// TIA Portal project "FullDemo" (V17)

(* hardware
DEVICE "S71500/ET200MP station_1"  S7-1500 station
   slot 0: "Rail_0"  Rack  6ES7 590-1***0-0AA0
   slot 0: "PM 70W 120/230VAC"  PM 70W 120/230VAC  6EP1332-4BA00
   slot 1: "S7-1500"  CPU 1513F-1 PN  6ES7 513-1FL01-0AB0  V2.0
      slot 3: "CPU display_1"  6ES7591-1AA00-0AA0
   slot 2: "DI 32x24VDC HF_1"  DI 32x24VDC HF  6ES7 521-1BL00-0AB0  V2.0
   slot 3: "DQ 32x24VDC/0.5A ST_1"  DQ 32x24VDC/0.5A ST  6ES7 522-1BL00-0AB0  V2.0
   slot 4: "AI 8xU/I/RTD/TC ST_1"  AI 8xU/I/RTD/TC ST  6ES7 531-7KF00-0AB0  V2.0
*)

// ===== PLC "S7-1500"  CPU 1513F-1 PN =====
// protected blocks, not shown: "FC_Signal"

VAR_GLOBAL   // PLC tag table "Default tag table"
   "Clock_Byte" AT %MB10 : Byte;
   "Clock_10Hz" AT %M10.0 : Bool;
   "Clock_5Hz" AT %M10.1 : Bool;
   "Clock_2.5Hz" AT %M10.2 : Bool;
   "Clock_2Hz" AT %M10.3 : Bool;
   "Clock_1.25Hz" AT %M10.4 : Bool;
   "Clock_1Hz" AT %M10.5 : Bool;
   "Clock_0.625Hz" AT %M10.6 : Bool;
   "Clock_0.5Hz" AT %M10.7 : Bool;
END_VAR

VAR_GLOBAL   // PLC tag table "Conveyor"
   "B_LB" AT %I4.0 : Bool;   // Lichtschranke / Light barrier
   "S_Bay1" AT %I4.1 : Bool;   // Taster Platz 1 / Momentary contact Bay 1
   "S_Bay2" AT %I4.2 : Bool;   // Taster Platz 2 / Momentary contact Bay 2
   "S_Bay3" AT %I4.3 : Bool;   // Taster Platz 3 / Momentary contact Bay 3
   "S_BayLB" AT %I4.4 : Bool;   // Taster Lichtschranken-Platz / Momentary contact Light barrier bay
   "B_Bay1" AT %I4.5 : Bool;   // Initiator Platz 1 / Proximity sensor Bay 1
   "B_Bay2" AT %I4.6 : Bool;   // Initiator Platz 2 / Proximity sensor Bay 2
   "B_Bay3" AT %I4.7 : Bool;   // Initiator Platz 3 / Proximity sensor Bay 3
   "P_Bay1" AT %Q4.1 : Bool;   // Meldeleuchte Platz 1 / Indicator light Bay 1
   "P_Bay2" AT %Q4.2 : Bool;   // Meldeleuchte Platz 2 / Indicator light Bay 2
   "P_Bay3" AT %Q4.3 : Bool;   // Meldeleuchte Platz 3 / Indicator light Bay 3
   "P_BayLB" AT %Q4.4 : Bool;   // Meldeleuchte Lichtschranken-Platz / Indicator light Light barrier bay
   "K_Right" AT %Q4.5 : Bool;   // Bandmotor Rechts / Run conveyor RIGHT
   "K_Left" AT %Q4.6 : Bool;   // Bandmotor Links / Run conveyor LEFT
   "P_Horn" AT %Q4.7 : Bool;   // Hupe / Horn
END_VAR

VAR_GLOBAL   // PLC tag table "My_Tags"
   "M_AuxLB" AT %M16.0 : Bool;   // Edge auxiliary memory bit Light barrier / Flanken-Hilfsmerker Lichtschranke
   "S_Fault3" AT %E0.6 : Bool;   // Schalter Störung 3 / S_Fault3
   "M_JogRight" AT %M16.2 : Bool;   // Merker Tippen Rechts / Memory bit Jog conveyor RIGHT
   "M_AutoRight" AT %M16.4 : Bool;   // Merker Auto Rechts / Memory bit Conveyor AUTO RIGHT
   "M_ConvFault" AT %M17.0 : Bool;   // Merker Bandlauf-Störung / Memory bit Conveyor fault
   "S_Acknowledge" AT %E0.7 : Bool;   // Taster Quittierung / S_Acknowledge
   "P_Operation" AT %A0.1 : Bool;   // Meldeleuchte Betrieb EIN / Indicator light Operation ON
   "P_Fault" AT %A0.7 : Bool;   // Anzeige Band-Störung / Indicator light for fault
   "M_AuxFault1" AT %M17.1 : Bool;   // Edge auxiliary memory bit Fault 1 / Flanken-Hilfsmerker Störung 1
   "P_Fault1" AT %A0.2 : Bool;   // Anzeige Störung 1 / Indicator light for fault1
   "P_Fault2" AT %A0.3 : Bool;   // Anzeige Störung 2 / Indicator light for fault2
   "S_Fault1" AT %E0.4 : Bool;   // Schalter Störung 1 / S_Fault1
   "S_Fault2" AT %E0.5 : Bool;   // Schalter Störung 2 / S_Fault2
   "P_Fault3" AT %A0.4 : Bool;   // Anzeige Störung 3 / Indicator light for fault3
   "M_AuxOpON" AT %M15.1 : Bool;   // Edge auxiliary memory bit Operation ON / Flanken-Hilfsmerker Anlage EIN
   "M_ActSetp" AT %M18.4 : Bool;   // Merker Ist-Stückzahl=Soll-Stückzah / Memory bit Actual- has reached Setpoint number
   "S_OperationON" AT %E0.1 : Bool;   // Taster Betrieb EIN / S_OperationON
   "S_OperationOFF" AT %E0.0 : Bool;   // Taster Betrieb AUS / S_OperationOFF
   "S_Right" AT %E0.2 : Bool;   // Taster Tippen Rechts / S_Right
   "S_Left" AT %E0.3 : Bool;   // Taster Tippen Links / S_Left
   "M_StorFault1" AT %M17.2 : Bool;   // Memory bit for storing Fault 1 / Merker Meldespeicher Störung 1
   "M_AuxFault2" AT %M17.3 : Bool;   // Edge auxiliary memory bit Fault 2 / Flanken-Hilfsmerker Störung 2
   "M_StorFault2" AT %M17.4 : Bool;   // Memory bit for storing Fault 2 / Merker Meldespeicher Störung 2
   "TOF-Timer-L" AT %M20.2 : Bool;
   "TOF-Timer-R" AT %M20.1 : Bool;
   "max_ConvFault" AT %M20.0 : Bool;
   "P_InitLeft" AT %A0.5 : Bool;
   "P_InitRight" AT %A0.6 : Bool;
   "S_Slider1" AT %IW10 : Word;
   "S_Slider2" AT %IW30 : Word;
END_VAR

VAR_GLOBAL CONSTANT   // PLC tag table "My_Tags"
   "const_maxTime" : Time := t#6s;   // max. Transportzeit / max. transport time
   "const_Setp" : UInt := 3;   // Sollwert / setpoint parts
END_VAR

VAR_GLOBAL   // PLC tag table "Drive"
   "StatusWordDrive" AT %EW60 : Word;
   "ActualSpeedDrive" AT %EW62 : Int;
   "ControlWordDrive" AT %AW60 : Word;
   "SetPointSpeedDrive" AT %AW62 : Int;
   "P_VoltageDisplay2" AT %AW34 : Word;
END_VAR

DATA_BLOCK "iDB_FB_FaultEvaluation"   // DB2
{ S7_Optimized_Access := 'TRUE' }
VERSION : 0.1
// stored: InstanceOfName FB_FaultEvaluation
"FB_FaultEvaluation"
BEGIN
END_DATA_BLOCK

DATA_BLOCK "iDB_FB_FaultEvaluation_2"   // DB3
{ S7_Optimized_Access := 'TRUE' }
VERSION : 0.1
// stored: InstanceOfName FB_FaultEvaluation
"FB_FaultEvaluation"
BEGIN
END_DATA_BLOCK

DATA_BLOCK "DB_Memory"   // DB8
{ S7_Optimized_Access := 'TRUE' }
VERSION : 0.1
   VAR
      Init_Right : Bool;
      Init_Left : Bool;
   END_VAR
   VAR RETAIN
      Operation : Bool;
   END_VAR
BEGIN
END_DATA_BLOCK

DATA_BLOCK "iDB_FB_Count"   // DB18
{ S7_Optimized_Access := 'TRUE' }
VERSION : 0.1
// stored: InstanceOfName FB_Count
"FB_Count"
BEGIN
END_DATA_BLOCK

DATA_BLOCK "iDB_FB_CountADD"   // DB19
{ S7_Optimized_Access := 'TRUE' }
VERSION : 0.1
// stored: InstanceOfName FB_CountADD
"FB_CountADD"
BEGIN
END_DATA_BLOCK

DATA_BLOCK "DB_OP"   // DB99
{ S7_Optimized_Access := 'TRUE' }
VERSION : 0.1
   VAR RETAIN
      OperationOFF : Bool;   // Anlage AUS (HMI) / Operation OFF
      OperationON : Bool;   // Anlage EIN (HMI) / Operation ON
      JogRight : Bool;   // Bandmotor Tippen Rechts / Jog conveyor motor right
      JogLeft : Bool;   // Bandmotor Tippen Links / Jog conveyor motor left
      AcknFault : Bool;   // Band-Störung quittieren / Acknowlwdge faults
      ActNo : UInt;   // Ist-Stückzahl / Actual quantity of parts
      SetpNo : UInt := 6;   // Soll-Stückzahl / Setpoint quantity of parts
   END_VAR
BEGIN
END_DATA_BLOCK

// folder: System blocks/Program resources

DATA_BLOCK "iDB_IEC_Timer_1"   // DB1
{ S7_Optimized_Access := 'TRUE' }
AUTHOR : Simatic
FAMILY : IEC
NAME : IEC_TMR
VERSION : 1.0
// stored: InstanceOfName IEC_TIMER
"IEC_TIMER"
BEGIN
END_DATA_BLOCK

DATA_BLOCK "iDB_IEC_Counter_1"   // DB4
{ S7_Optimized_Access := 'TRUE' }
AUTHOR : Simatic
FAMILY : IEC
NAME : UCNTR
VERSION : 1.2
// stored: InstanceOfName IEC_UCOUNTER
"IEC_UCOUNTER"
BEGIN
END_DATA_BLOCK

DATA_BLOCK "IEC_Counter_0_DB"   // DB5
{ S7_Optimized_Access := 'TRUE' }
AUTHOR : Simatic
FAMILY : IEC
NAME : CNTR
VERSION : 1.0
// stored: InstanceOfName IEC_COUNTER
"IEC_COUNTER"
BEGIN
END_DATA_BLOCK

DATA_BLOCK "IEC_Timer_0_DB"   // DB6
{ S7_Optimized_Access := 'TRUE' }
AUTHOR : Simatic
FAMILY : IEC
NAME : IEC_TMR
VERSION : 1.0
// stored: InstanceOfName IEC_TIMER
"IEC_TIMER"
BEGIN
END_DATA_BLOCK

DATA_BLOCK "IEC_Timer_1_DB"   // DB7
{ S7_Optimized_Access := 'TRUE' }
AUTHOR : Simatic
FAMILY : IEC
NAME : IEC_TMR
VERSION : 1.0
// stored: InstanceOfName IEC_TIMER
"IEC_TIMER"
BEGIN
END_DATA_BLOCK

// folder: (top level)

FUNCTION_BLOCK "FB_Count"   // FB18, LAD
{ S7_Optimized_Access := 'TRUE' }
VERSION : 0.1
   VAR_INPUT
      LB : Bool;
      Reset : Bool;
      Operation : Bool;
      Setp : UInt;
   END_VAR
   VAR_OUTPUT
      ActSetp : Bool;
   END_VAR
   VAR_IN_OUT
      Act : UInt;
   END_VAR
   VAR
      PosEdgeLB : Bool;
      PosEdgeOp : Bool;
   END_VAR
   VAR_TEMP   // added for the SCL form of the ladder/FBD networks
      _w1 : Bool;
   END_VAR
BEGIN

REGION Network 1: Count parts / Zählen der transportieren Teile
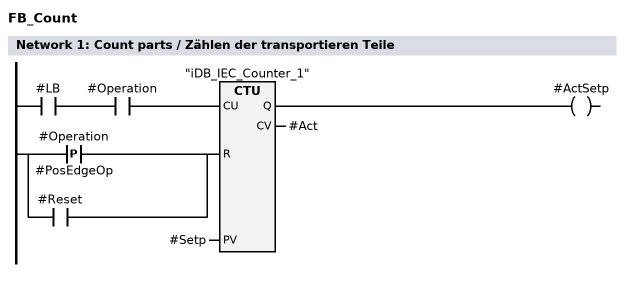
   #_w1 := #Operation AND NOT #PosEdgeOp;   // rising edge of #Operation
   #PosEdgeOp := #Operation;
   "iDB_IEC_Counter_1".CTU(CU := #LB AND #Operation, R := #_w1 OR #Reset, PV := #Setp, CV => #Act);
   #ActSetp := "iDB_IEC_Counter_1".Q;
END_REGION
END_FUNCTION_BLOCK

FUNCTION_BLOCK "FB_CountADD"   // FB19, LAD
{ S7_Optimized_Access := 'TRUE' }
VERSION : 0.1
   VAR_INPUT
      LB : Bool;
      Reset : Bool;
      Operation : Bool;
   END_VAR
   VAR_OUTPUT
      ActSetp : Bool;
   END_VAR
   VAR
      PosEdge : Bool;
      ActNo : UInt;
   END_VAR
   VAR CONSTANT
      const_Setp : UInt := 3;
   END_VAR
   VAR_TEMP   // added for the SCL form of the ladder/FBD networks
      _w1 : Bool;
   END_VAR
BEGIN

REGION Network 1: Reset Counter / Zähler rücksetzen
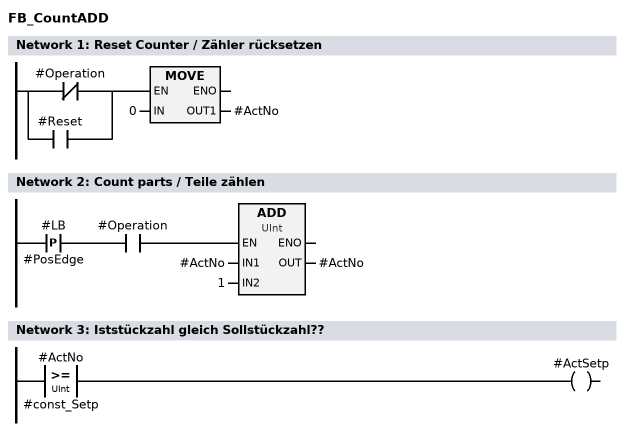
   RUNG wire#powerrail
      I_Contact( #Operation )
      wire#w1
      Move(in := 0, out1 => #ActNo)
   END_RUNG
   RUNG wire#powerrail
      Contact( #Reset )
   END_RUNG wire#w1
   // the same network as SCL:
   IF NOT #Operation OR #Reset THEN #ActNo := 0; END_IF;
END_REGION

REGION Network 2: Count parts / Teile zählen
   RUNG wire#powerrail
      P_Contact(operand := #LB, bit := #PosEdge)
      Contact( #Operation )
      { S7_Templates := "SrcType := UInt" } Add(in1 := #ActNo, in2 := 1, out => #ActNo)
   END_RUNG
   // the same network as SCL:
   #_w1 := #LB AND NOT #PosEdge;   // rising edge of #LB
   #PosEdge := #LB;
   IF #_w1 AND #Operation THEN #ActNo := #ActNo + 1; END_IF;
END_REGION

REGION Network 3: Iststückzahl gleich Sollstückzahl??
   RUNG wire#powerrail
      { S7_Templates := "SrcType := UInt" } GE_Contact(in1 := #ActNo, in2 := #const_Setp)
      Coil( #ActSetp )
   END_RUNG
   // the same network as SCL:
   #ActSetp := #ActNo >= #const_Setp;
END_REGION
END_FUNCTION_BLOCK

FUNCTION_BLOCK "FB_FaultEvaluation"   // FB20, LAD
{ S7_Optimized_Access := 'TRUE' }
VERSION : 0.1
   VAR_INPUT
      FaultInput : Bool;
      FlashFreq : Bool;
      Acknowledge : Bool;
   END_VAR
   VAR_OUTPUT
      Display : Bool;
   END_VAR
   VAR
      StoredFault : Bool;
      EdgeMemory : Bool;
   END_VAR
   VAR_TEMP   // added for the SCL form of the ladder/FBD networks
      _w1 : Bool;
   END_VAR
BEGIN

REGION Network 1: Fault evaluation / Störungsauswertung
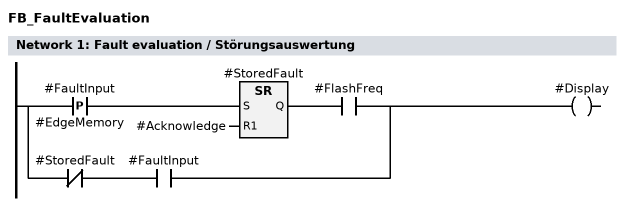
   RUNG wire#powerrail
      P_Contact(operand := #FaultInput, bit := #EdgeMemory)
      S_SR(operand := #StoredFault, r1 := #Acknowledge)
      Contact( #FlashFreq )
      wire#w1
      Coil( #Display )
   END_RUNG
   RUNG wire#powerrail
      I_Contact( #StoredFault )
      Contact( #FaultInput )
   END_RUNG wire#w1
   // the same network as SCL:
   #_w1 := #FaultInput AND NOT #EdgeMemory;   // rising edge of #FaultInput
   #EdgeMemory := #FaultInput;
   IF #_w1 THEN
       #StoredFault := TRUE;   // SR flip-flop
   END_IF;
   IF #Acknowledge THEN #StoredFault := FALSE; END_IF;
   #Display := (#StoredFault AND #FlashFreq) OR (NOT #StoredFault AND #FaultInput);
END_REGION
END_FUNCTION_BLOCK

FUNCTION "FC_Mode" : Void   // FC15, LAD
{ S7_Optimized_Access := 'TRUE' }
VERSION : 0.1
BEGIN

REGION Network 1: Meldeleuchte Betrieb EIN / Operation ON/OFF
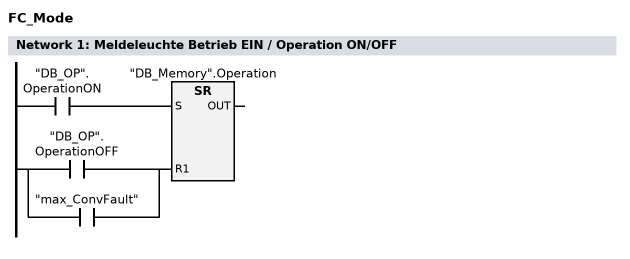
   RUNG wire#powerrail
      Contact( "DB_OP".OperationON )
      S_SR(operand := "DB_Memory".Operation, r1 := wire#w1)
   END_RUNG
   RUNG wire#powerrail
      Contact( "DB_OP".OperationOFF )
   END_RUNG wire#w1
   RUNG wire#powerrail
      Contact( "max_ConvFault" )
   END_RUNG wire#w1
   // the same network as SCL:
   IF "DB_OP".OperationON THEN
       "DB_Memory".Operation := TRUE;   // SR flip-flop
   END_IF;
   IF "DB_OP".OperationOFF OR "max_ConvFault" THEN "DB_Memory".Operation := FALSE; END_IF;
END_REGION
END_FUNCTION

FUNCTION "FC_Conveyor" : Void   // FC16, LAD
{ S7_Optimized_Access := 'TRUE' }
VERSION : 0.1
   VAR_TEMP   // added for the SCL form of the ladder/FBD networks
      _w1 : Bool;
   END_VAR
BEGIN

REGION Network 1: Tippen rechts / Memory bit Jog conveyor RIGHT
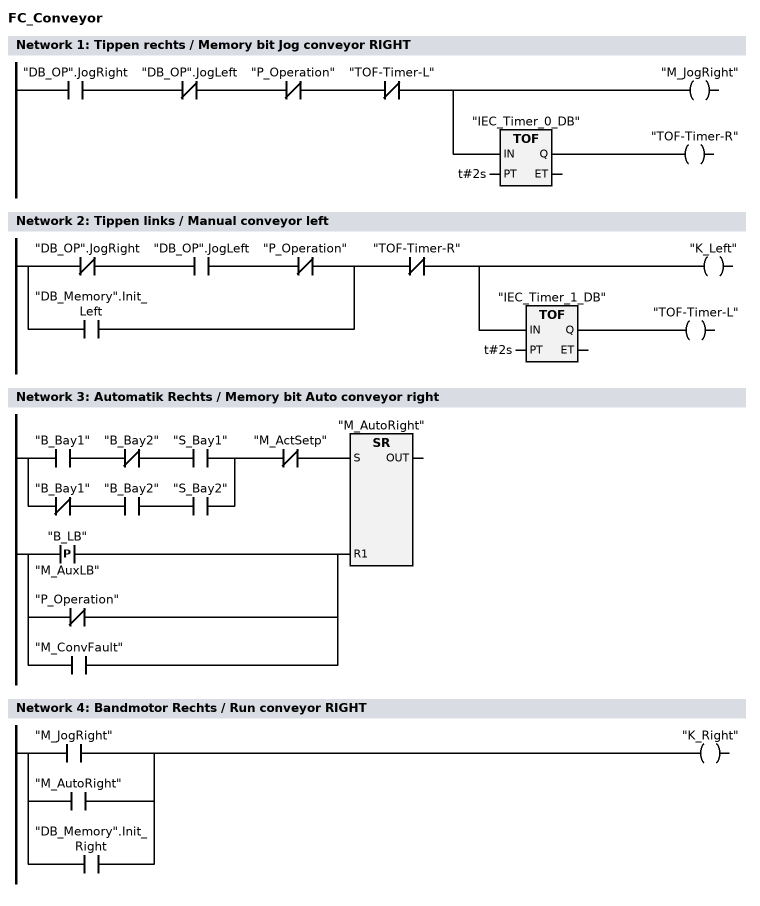
   "M_JogRight" := "DB_OP".JogRight AND NOT "DB_OP".JogLeft AND NOT "P_Operation" AND NOT "TOF-Timer-L";
   "IEC_Timer_0_DB".TOF(IN := "M_JogRight", PT := t#2s);
   "TOF-Timer-R" := "IEC_Timer_0_DB".Q;
END_REGION

REGION Network 2: Tippen links / Manual conveyor left
   "K_Left" := ((NOT "DB_OP".JogRight AND "DB_OP".JogLeft AND NOT "P_Operation") OR "DB_Memory".Init_Left) AND NOT "TOF-Timer-R";
   "IEC_Timer_1_DB".TOF(IN := "K_Left", PT := t#2s);
   "TOF-Timer-L" := "IEC_Timer_1_DB".Q;
END_REGION

REGION Network 3: Automatik Rechts / Memory bit Auto conveyor right
   RUNG wire#powerrail
      Contact( "B_Bay1" )
      I_Contact( "B_Bay2" )
      Contact( "S_Bay1" )
      wire#w1
      I_Contact( "M_ActSetp" )
      S_SR(operand := "M_AutoRight", r1 := wire#w2)
   END_RUNG
   RUNG wire#powerrail
      I_Contact( "B_Bay1" )
      Contact( "B_Bay2" )
      Contact( "S_Bay2" )
   END_RUNG wire#w1
   RUNG wire#powerrail
      P_Contact(operand := "B_LB", bit := "M_AuxLB")
   END_RUNG wire#w2
   RUNG wire#powerrail
      I_Contact( "P_Operation" )
   END_RUNG wire#w2
   RUNG wire#powerrail
      Contact( "M_ConvFault" )
   END_RUNG wire#w2
   // the same network as SCL:
   #_w1 := "B_LB" AND NOT "M_AuxLB";   // rising edge of "B_LB"
   "M_AuxLB" := "B_LB";
   IF (("B_Bay1" AND NOT "B_Bay2" AND "S_Bay1") OR (NOT "B_Bay1" AND "B_Bay2" AND "S_Bay2")) AND NOT "M_ActSetp" THEN
       "M_AutoRight" := TRUE;   // SR flip-flop
   END_IF;
   IF #_w1 OR NOT "P_Operation" OR "M_ConvFault" THEN "M_AutoRight" := FALSE; END_IF;
END_REGION

REGION Network 4: Bandmotor Rechts / Run conveyor RIGHT
   RUNG wire#powerrail
      Contact( "M_JogRight" )
      wire#w1
      Coil( "K_Right" )
   END_RUNG
   RUNG wire#powerrail
      Contact( "M_AutoRight" )
   END_RUNG wire#w1
   RUNG wire#powerrail
      Contact( "DB_Memory".Init_Right )
   END_RUNG wire#w1
   // the same network as SCL:
   "K_Right" := "M_JogRight" OR "M_AutoRight" OR "DB_Memory".Init_Right;
END_REGION
END_FUNCTION

FUNCTION "FC_Fault" : Void   // FC17, LAD
{ S7_Optimized_Access := 'TRUE' }
VERSION : 0.1
BEGIN

REGION Network 1: Band-Störung
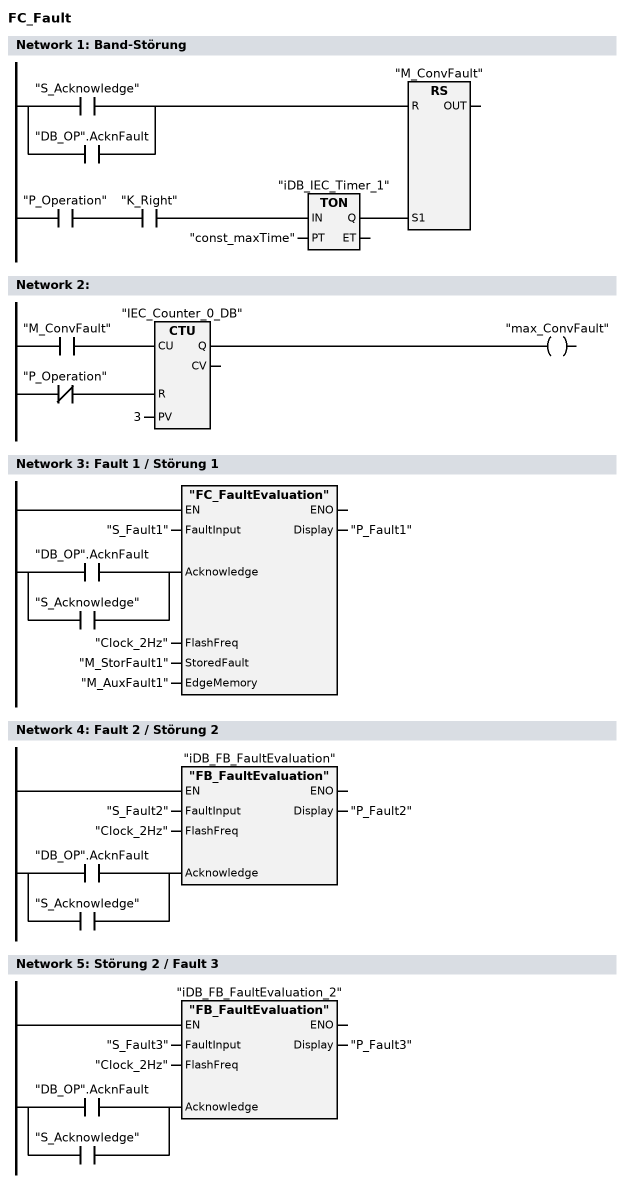
   "iDB_IEC_Timer_1".TON(IN := "P_Operation" AND "K_Right", PT := "const_maxTime");
   IF "S_Acknowledge" OR "DB_OP".AcknFault THEN
       "M_ConvFault" := FALSE;   // RS flip-flop
   END_IF;
   IF "iDB_IEC_Timer_1".Q THEN "M_ConvFault" := TRUE; END_IF;
END_REGION

REGION Network 2
   "IEC_Counter_0_DB".CTU(CU := "M_ConvFault", R := NOT "P_Operation", PV := 3);
   "max_ConvFault" := "IEC_Counter_0_DB".Q;
END_REGION

REGION Network 3: Fault 1 / Störung 1
   RUNG wire#powerrail
      "FC_FaultEvaluation"(Acknowledge := wire#w1, FaultInput := "S_Fault1", FlashFreq := "Clock_2Hz", StoredFault := "M_StorFault1", EdgeMemory := "M_AuxFault1", Display => "P_Fault1")
   END_RUNG
   RUNG wire#powerrail
      Contact( "DB_OP".AcknFault )
   END_RUNG wire#w1
   RUNG wire#powerrail
      Contact( "S_Acknowledge" )
   END_RUNG wire#w1
   // the same network as SCL:
   "FC_FaultEvaluation"(FaultInput := "S_Fault1",
                        Acknowledge := "DB_OP".AcknFault OR "S_Acknowledge",
                        FlashFreq := "Clock_2Hz",
                        StoredFault := "M_StorFault1",
                        EdgeMemory := "M_AuxFault1",
                        Display => "P_Fault1");
END_REGION

REGION Network 4: Fault 2 / Störung 2
   RUNG wire#powerrail
      "iDB_FB_FaultEvaluation"(Acknowledge := wire#w1, FaultInput := "S_Fault2", FlashFreq := "Clock_2Hz", Display => "P_Fault2")
   END_RUNG
   RUNG wire#powerrail
      Contact( "DB_OP".AcknFault )
   END_RUNG wire#w1
   RUNG wire#powerrail
      Contact( "S_Acknowledge" )
   END_RUNG wire#w1
   // the same network as SCL:
   "iDB_FB_FaultEvaluation"(FaultInput := "S_Fault2",   // "FB_FaultEvaluation"
                           FlashFreq := "Clock_2Hz",
                           Acknowledge := "DB_OP".AcknFault OR "S_Acknowledge",
                           Display => "P_Fault2");
END_REGION

REGION Network 5: Störung 2 / Fault 3
   RUNG wire#powerrail
      "iDB_FB_FaultEvaluation_2"(Acknowledge := wire#w1, FaultInput := "S_Fault3", FlashFreq := "Clock_2Hz", Display => "P_Fault3")
   END_RUNG
   RUNG wire#powerrail
      Contact( "DB_OP".AcknFault )
   END_RUNG wire#w1
   RUNG wire#powerrail
      Contact( "S_Acknowledge" )
   END_RUNG wire#w1
   // the same network as SCL:
   "iDB_FB_FaultEvaluation_2"(FaultInput := "S_Fault3",   // "FB_FaultEvaluation"
                           FlashFreq := "Clock_2Hz",
                           Acknowledge := "DB_OP".AcknFault OR "S_Acknowledge",
                           Display => "P_Fault3");
END_REGION
END_FUNCTION

FUNCTION "FC_FaultEvaluation" : Void   // FC20, LAD
{ S7_Optimized_Access := 'TRUE' }
VERSION : 0.1
   VAR_INPUT
      FaultInput : Bool;
      Acknowledge : Bool;
      FlashFreq : Bool;
   END_VAR
   VAR_OUTPUT
      Display : Bool;
   END_VAR
   VAR_IN_OUT
      StoredFault : Bool;
      EdgeMemory : Bool;
   END_VAR
   VAR_TEMP   // added for the SCL form of the ladder/FBD networks
      _w1 : Bool;
   END_VAR
BEGIN

REGION Network 1: Fault evaluation / Störungsauswertung
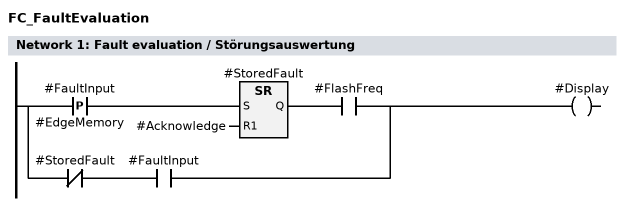
   RUNG wire#powerrail
      P_Contact(operand := #FaultInput, bit := #EdgeMemory)
      S_SR(operand := #StoredFault, r1 := #Acknowledge)
      Contact( #FlashFreq )
      wire#w1
      Coil( #Display )
   END_RUNG
   RUNG wire#powerrail
      I_Contact( #StoredFault )
      Contact( #FaultInput )
   END_RUNG wire#w1
   // the same network as SCL:
   #_w1 := #FaultInput AND NOT #EdgeMemory;   // rising edge of #FaultInput
   #EdgeMemory := #FaultInput;
   IF #_w1 THEN
       #StoredFault := TRUE;   // SR flip-flop
   END_IF;
   IF #Acknowledge THEN #StoredFault := FALSE; END_IF;
   #Display := (#StoredFault AND #FlashFreq) OR (NOT #StoredFault AND #FaultInput);
END_REGION
END_FUNCTION

FUNCTION "FC_Drive" : Void   // FC120, LAD
TITLE = Antrieb ansteuern
{ S7_Optimized_Access := 'TRUE' }
VERSION : 0.1
   VAR_TEMP
      temp_Percent : Real;
   END_VAR
   VAR_TEMP   // added for the SCL form of the ladder/FBD networks
      _w1 : Bool;
   END_VAR
BEGIN

REGION Network 1: Spannungswert anzeigen
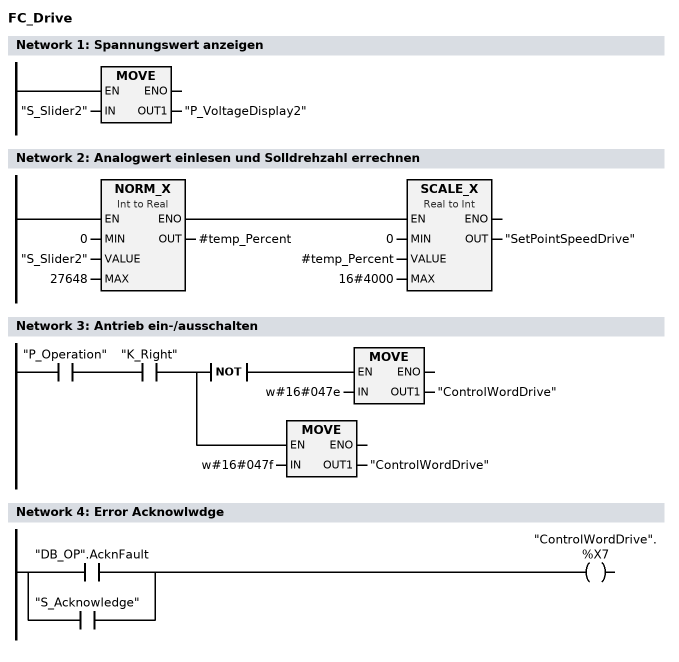
   RUNG wire#powerrail
      Move(in := "S_Slider2", out1 => "P_VoltageDisplay2")
   END_RUNG
   // the same network as SCL:
   "P_VoltageDisplay2" := "S_Slider2";
END_REGION

REGION Network 2: Analogwert einlesen und Solldrehzahl errechnen
   RUNG wire#powerrail
      { S7_Templates := "[SrcType := Int, DestType := Real]" } Normalize(min := 0, value := "S_Slider2", max := 27648, out => #temp_Percent)
      { S7_Templates := "[SrcType := Real, DestType := Int]" } Scale(min := 0, value := #temp_Percent, max := 16#4000, out => "SetPointSpeedDrive")
   END_RUNG
   // the same network as SCL:
   #temp_Percent := NORM_X(MIN := 0, VALUE := "S_Slider2", MAX := 27648);
   "SetPointSpeedDrive" := SCALE_X(MIN := 0, VALUE := #temp_Percent, MAX := 16#4000);
END_REGION

REGION Network 3: Antrieb ein-/ausschalten
   RUNG wire#powerrail
      Contact( "P_Operation" )
      Contact( "K_Right" )
      wire#w1
      Not()
      { S7_GenerateENO := "TRUE" } Move(in := w#16#047e, out1 => "ControlWordDrive")
   END_RUNG
   RUNG wire#w1
      { S7_GenerateENO := "TRUE" } Move(in := w#16#047f, out1 => "ControlWordDrive")
   END_RUNG
   // the same network as SCL:
   #_w1 := "P_Operation" AND "K_Right";
   IF NOT #_w1 THEN "ControlWordDrive" := w#16#047e; END_IF;
   IF #_w1 THEN "ControlWordDrive" := w#16#047f; END_IF;
END_REGION

REGION Network 4: Error Acknowlwdge
   RUNG wire#powerrail
      Contact( "DB_OP".AcknFault )
      wire#w1
      Coil( "ControlWordDrive".%X7 )
   END_RUNG
   RUNG wire#powerrail
      Contact( "S_Acknowledge" )
   END_RUNG wire#w1
   // the same network as SCL:
   "ControlWordDrive".%X7 := "DB_OP".AcknFault OR "S_Acknowledge";
END_REGION
END_FUNCTION

ORGANIZATION_BLOCK "OB_Cycle"   // OB1, LAD, ProgramCycle
TITLE = "Main Program Sweep (Cycle)"
{ S7_Optimized_Access := 'TRUE' }
VERSION : 0.1
   VAR_INPUT
      Initial_Call : Bool;   // Initial call of this OB
      Remanence : Bool;   // =True, if remanent data are available
   END_VAR
BEGIN

REGION Network 1: Operation mode
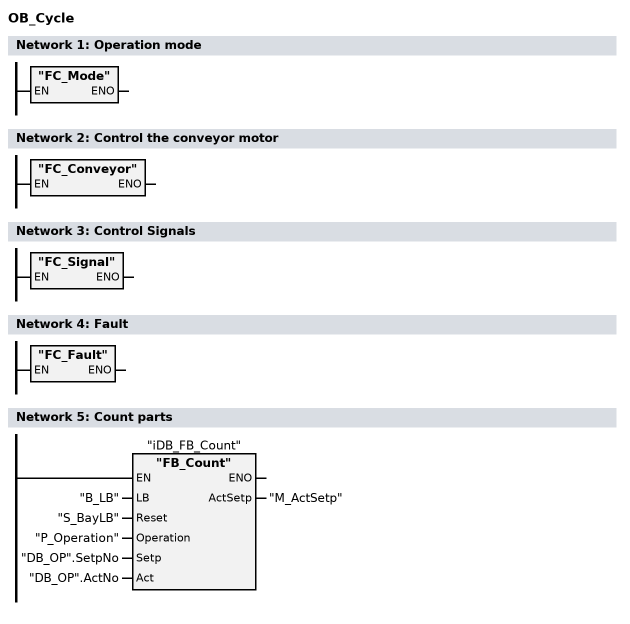
   RUNG wire#powerrail
      "FC_Mode"()
   END_RUNG
   // the same network as SCL:
   "FC_Mode"();
END_REGION

REGION Network 2: Control the conveyor motor
   RUNG wire#powerrail
      "FC_Conveyor"()
   END_RUNG
   // the same network as SCL:
   "FC_Conveyor"();
END_REGION

REGION Network 3: Control Signals
   RUNG wire#powerrail
      "FC_Signal"()
   END_RUNG
   // the same network as SCL:
   "FC_Signal"();
END_REGION

REGION Network 4: Fault
   RUNG wire#powerrail
      "FC_Fault"()
   END_RUNG
   // the same network as SCL:
   "FC_Fault"();
END_REGION

REGION Network 5: Count parts
   RUNG wire#powerrail
      "iDB_FB_Count"(LB := "B_LB", Reset := "S_BayLB", Operation := "P_Operation", Setp := "DB_OP".SetpNo, Act := "DB_OP".ActNo, ActSetp => "M_ActSetp")
   END_RUNG
   // the same network as SCL:
   "iDB_FB_Count"(LB := "B_LB",   // "FB_Count"
                  Reset := "S_BayLB",
                  Operation := "P_Operation",
                  Setp := "DB_OP".SetpNo,
                  Act := "DB_OP".ActNo,
                  ActSetp => "M_ActSetp");
END_REGION
END_ORGANIZATION_BLOCK

ORGANIZATION_BLOCK "OB_Time delay interrupt_1"   // OB20, LAD, TimeDelayInterrupt
TITLE = Time dalay interrupt
{ S7_Optimized_Access := 'TRUE' }
VERSION : 0.1
   VAR_INPUT
      Sign : Word;   // Identifier input (SIGN) passed to triggering call of SRT_DINT
   END_VAR
BEGIN

REGION Network 1: Inittialisierung Links Stop
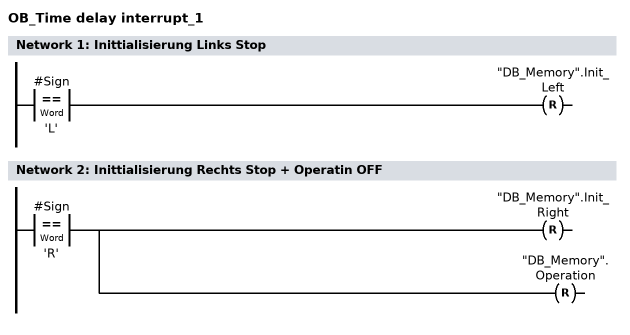
   RUNG wire#powerrail
      { S7_Templates := "SrcType := Word" } EQ_Contact(in1 := #Sign, in2 := 'L')
      R_Coil( "DB_Memory".Init_Left )
   END_RUNG
   // the same network as SCL:
   IF #Sign = 'L' THEN "DB_Memory".Init_Left := FALSE; END_IF;
END_REGION

REGION Network 2: Inittialisierung Rechts Stop + Operatin OFF
   RUNG wire#powerrail
      { S7_Templates := "SrcType := Word" } EQ_Contact(in1 := #Sign, in2 := 'R')
      wire#w1
      R_Coil( "DB_Memory".Init_Right )
   END_RUNG
   RUNG wire#w1
      R_Coil( "DB_Memory".Operation )
   END_RUNG
   // the same network as SCL:
   IF #Sign = 'R' THEN
       "DB_Memory".Init_Right := FALSE;
       "DB_Memory".Operation := FALSE;
   END_IF;
END_REGION
END_ORGANIZATION_BLOCK

ORGANIZATION_BLOCK "Cyclic interrupt_Trace"   // OB30, LAD, CyclicInterrupt
{ S7_Optimized_Access := 'TRUE' }
VERSION : 0.1
   VAR_INPUT
      Initial_Call : Bool;   // Initial call of this OB
      Event_Count : Int;   // Events discarded
   END_VAR
BEGIN
END_ORGANIZATION_BLOCK

ORGANIZATION_BLOCK "OB_Startup_1"   // OB100, LAD, Startup
TITLE = "Complete Restart"
{ S7_Optimized_Access := 'TRUE' }
VERSION : 0.1
   VAR_INPUT
      LostRetentive : Bool;   // True if retentive data are lost
      LostRTC : Bool;   // True if date and time are lost
   END_VAR
   VAR_TEMP
      ret_V : Int;
      Startinfo : Word;
   END_VAR
   VAR CONSTANT
      constInitTime : Time := T#5s;
   END_VAR
BEGIN

REGION Network 1: Inititialisierung links starten / start initialisation left
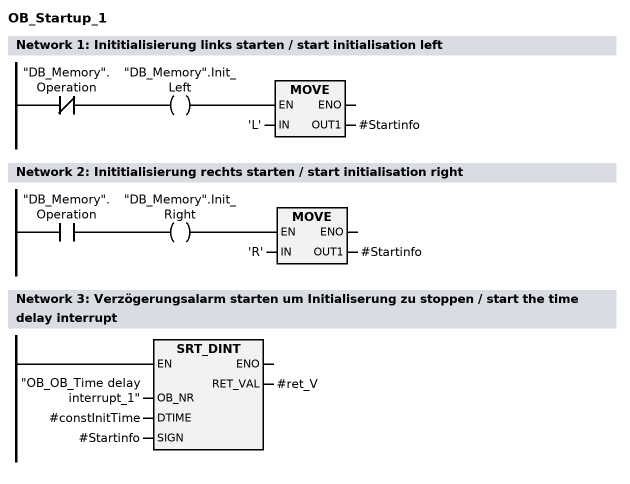
   RUNG wire#powerrail
      I_Contact( "DB_Memory".Operation )
      Coil( "DB_Memory".Init_Left )
      Move(in := 'L', out1 => #Startinfo)
   END_RUNG
   // the same network as SCL:
   "DB_Memory".Init_Left := NOT "DB_Memory".Operation;
   IF NOT "DB_Memory".Operation THEN #Startinfo := 'L'; END_IF;
END_REGION

REGION Network 2: Inititialisierung rechts starten / start initialisation right
   RUNG wire#powerrail
      Contact( "DB_Memory".Operation )
      Coil( "DB_Memory".Init_Right )
      Move(in := 'R', out1 => #Startinfo)
   END_RUNG
   // the same network as SCL:
   "DB_Memory".Init_Right := "DB_Memory".Operation;
   IF "DB_Memory".Operation THEN #Startinfo := 'R'; END_IF;
END_REGION

REGION Network 3: Verzögerungsalarm starten um Initialiserung zu stoppen / start the time delay interrupt
   #ret_V := SRT_DINT(OB_NR := "OB_OB_Time delay interrupt_1", DTIME := #constInitTime, SIGN := #Startinfo);
END_REGION
END_ORGANIZATION_BLOCK

ORGANIZATION_BLOCK "OB_Cycle_Drive"   // OB123, LAD, ProgramCycle
TITLE = "Main Program Sweep (Cycle)"
{ S7_Optimized_Access := 'TRUE' }
VERSION : 0.1
   VAR_INPUT
      Initial_Call : Bool;   // Initial call of this OB
      Remanence : Bool;   // =True, if remanent data are available
   END_VAR
BEGIN

REGION Network 1
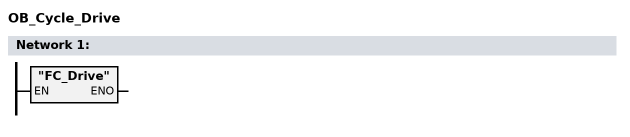
   RUNG wire#powerrail
      "FC_Drive"()
   END_RUNG
   // the same network as SCL:
   "FC_Drive"();
END_REGION
END_ORGANIZATION_BLOCK